// TIA Portal V17 export
// export: Created 2024-01-30T08:49:16.9839583Z, ExportSetting WithDefaults, DisplayName Totally Integrated Automation Portal, DisplayVersion V17 Update 6, DisplayName TIA Portal Openness, DisplayVersion V17 Update 6, DisplayName TIA Portal Version Control Interface, DisplayVersion V17, DisplayName STEP 7 Professional, DisplayVersion V17 Update 6, DisplayName STEP 7 Safety, DisplayVersion V17 Update 6, DisplayName WinCC Advanced, DisplayVersion V17 Update 6
VAR_GLOBAL   // PLC tag table "LK_G5000"
   TO_LKG5000_CTRL AT %Q339.0 : "UDT_LKG5000_RS232_SEND";
   FROM_LKG5000_CTRL AT %I11.0 : "UDT_LKG5000_RS232_RCV";
   SEND_DATA AT %Q344.0 : "UDT_RS232_SEND_DATA";
   RCV_DATA AT %I351.0 : "UDT_RS232_RCV_DATA";
END_VAR
